(* Logix 5000 project; controller Project vendor 1 type 14 code 92 rev 37.11; software revision 37.00 *)

TASK MainTask (continuous, watchdog 500 ms) : MainProgram, new_test_program

MODULES
   Local : vendor 1 type 14 code 92 (ICP 0, rev 37.11)
END_MODULES

VAR_GLOBAL   (* controller tags *)
   x7 : BOOL;
END_VAR

PROGRAM MainProgram   (* main routine MainRoutine *)
VAR
   input : BOOL;
   next_input : BOOL;
   output_1 : BOOL;
END_VAR

ROUTINE MainRoutine   (* ladder *)
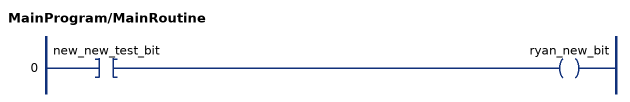
   0: XIC(new_new_test_bit)OTE(ryan_new_bit);
END_ROUTINE
END_PROGRAM

PROGRAM new_test_program   (* main routine new_test_routine *)
// making changes

ROUTINE new_test_routine   (* ladder *)
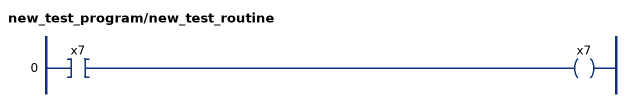
   0: XIC(x7)OTE(x7);
END_ROUTINE
END_PROGRAM
